// LS Electric XG5000 project: mecomhmi_plc
// PLC LSPLC

PROGRAM NewProgram (task: 스캔 프로그램)

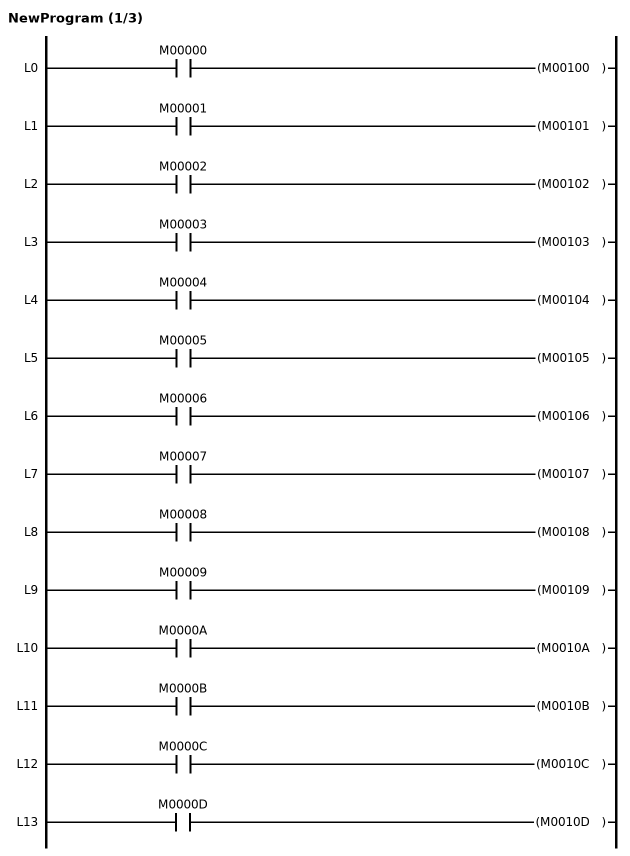
; L0
LOAD      M00000
OUT       M00100
; L1
LOAD      M00001
OUT       M00101
; L2
LOAD      M00002
OUT       M00102
; L3
LOAD      M00003
OUT       M00103
; L4
LOAD      M00004
OUT       M00104
; L5
LOAD      M00005
OUT       M00105
; L6
LOAD      M00006
OUT       M00106
; L7
LOAD      M00007
OUT       M00107
; L8
LOAD      M00008
OUT       M00108
; L9
LOAD      M00009
OUT       M00109
; L10
LOAD      M0000A
OUT       M0010A
; L11
LOAD      M0000B
OUT       M0010B
; L12
LOAD      M0000C
OUT       M0010C
; L13
LOAD      M0000D
OUT       M0010D

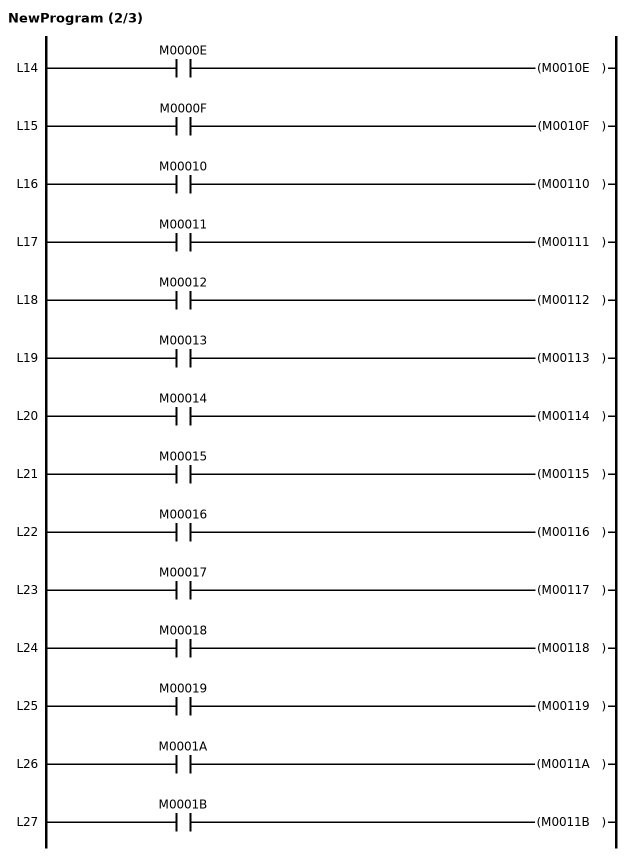
; L14
LOAD      M0000E
OUT       M0010E
; L15
LOAD      M0000F
OUT       M0010F
; L16
LOAD      M00010
OUT       M00110
; L17
LOAD      M00011
OUT       M00111
; L18
LOAD      M00012
OUT       M00112
; L19
LOAD      M00013
OUT       M00113
; L20
LOAD      M00014
OUT       M00114
; L21
LOAD      M00015
OUT       M00115
; L22
LOAD      M00016
OUT       M00116
; L23
LOAD      M00017
OUT       M00117
; L24
LOAD      M00018
OUT       M00118
; L25
LOAD      M00019
OUT       M00119
; L26
LOAD      M0001A
OUT       M0011A
; L27
LOAD      M0001B
OUT       M0011B

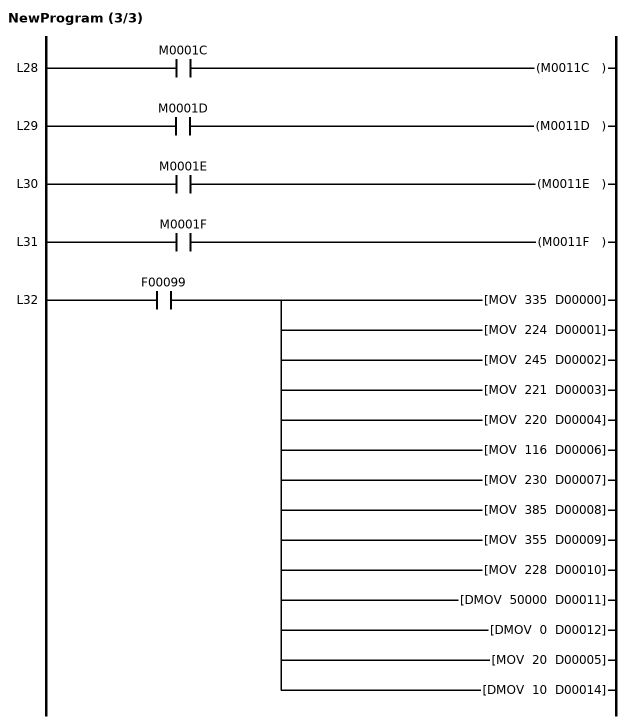
; L28
LOAD      M0001C
OUT       M0011C
; L29
LOAD      M0001D
OUT       M0011D
; L30
LOAD      M0001E
OUT       M0011E
; L31
LOAD      M0001F
OUT       M0011F
; L32
LOAD      F00099
MOV       335 D00000
MOV       224 D00001
MOV       245 D00002
MOV       221 D00003
MOV       220 D00004
MOV       116 D00006
MOV       230 D00007
MOV       385 D00008
MOV       355 D00009
MOV       228 D00010
DMOV      50000 D00011
DMOV      0 D00012
MOV       20 D00005
DMOV      10 D00014